_CFC_ (* Continuous Function Chart, elements in execution order *)
#0 INT_TO_REAL(SCHU_P2_4_TE2_AI2)
#1 DIV(#0, 10)
#2 SCHU_P2_4_TE2_VN <= #1
#3 I_GT_TE:ISTOK_GT(dost: TRUE, x: #1, ust: SCHU_P2_4_TE_HIGHLIMIT, shkal: -, gist: 1)
#4 I_LT_TE:ISTOK_LT(dost: TRUE, x: #1, ust: SCHU_P2_4_TE_LOWLIMIT, shkal: -, gist: 1)
#5 OR(#3.Xb, #4.Xm)
#6 TON_DOST:TON(IN: NOT #5, PT: T#10s)
#7 SCHU_P2_4_TE2_DOST <= #6.Q
#8 fb_SCHU_P2_4_TE2_M_UST:ISTOK_LT(dost: #6.Q, x: #1, ust: SCHU_P2_4_TE2_UST, shkal: -, gist: 5)
#9 SCHU_P2_4_TE2_M_UST <= #8.Xm
#10 SCHU_P2_4_TE2_B_UST <= #8.XmN
#11 SUB(SCHU_P2_4_TE2_ZASCH_OTKL, SCHU_P2_4_TE2_ZASCH)
#12 fb_SCHU_P2_4_TE2_M_ZASCH:ISTOK_LT(dost: #6.Q, x: #1, ust: SCHU_P2_4_TE2_ZASCH, shkal: -, gist: #11)
#13 SCHU_P2_4_TE2_M_ZASCH <= #12.Xm
#14 SCHU_P2_4_TE2_B_ZASCH <= #12.XmN
_END_CFC_
(* the same logic as Structured Text *)
_t112 := INT_TO_REAL(SCHU_P2_4_TE2_AI2) / 10;
SCHU_P2_4_TE2_VN := _t112;
I_GT_TE(dost := TRUE, x := _t112, ust := SCHU_P2_4_TE_HIGHLIMIT, gist := 1);
I_LT_TE(dost := TRUE, x := _t112, ust := SCHU_P2_4_TE_LOWLIMIT, gist := 1);
TON_DOST(IN := NOT (I_GT_TE.Xb OR I_LT_TE.Xm), PT := T#10s);
SCHU_P2_4_TE2_DOST := TON_DOST.Q;
fb_SCHU_P2_4_TE2_M_UST(dost := TON_DOST.Q, x := _t112, ust := SCHU_P2_4_TE2_UST, gist := 5);
SCHU_P2_4_TE2_M_UST := fb_SCHU_P2_4_TE2_M_UST.Xm;
SCHU_P2_4_TE2_B_UST := fb_SCHU_P2_4_TE2_M_UST.XmN;
fb_SCHU_P2_4_TE2_M_ZASCH(dost := TON_DOST.Q, x := _t112, ust := SCHU_P2_4_TE2_ZASCH, gist := SCHU_P2_4_TE2_ZASCH_OTKL - SCHU_P2_4_TE2_ZASCH);
SCHU_P2_4_TE2_M_ZASCH := fb_SCHU_P2_4_TE2_M_ZASCH.Xm;
SCHU_P2_4_TE2_B_ZASCH := fb_SCHU_P2_4_TE2_M_ZASCH.XmN;
END_PROGRAM

(* POU Input/AI/UE1_T, CFC *)
PROGRAM UE1_T
VAR
	fb_UE2_T: ISTOK_ANALOGVH;
	ofset: REAL;
	fb_UE2eqUST: ISTOK_EQ;
	fb_UE2_m_UST: ISTOK_LT;
	fb_UE2_b_UST: ISTOK_GT;
	enbleLimit: BOOL;
END_VAR
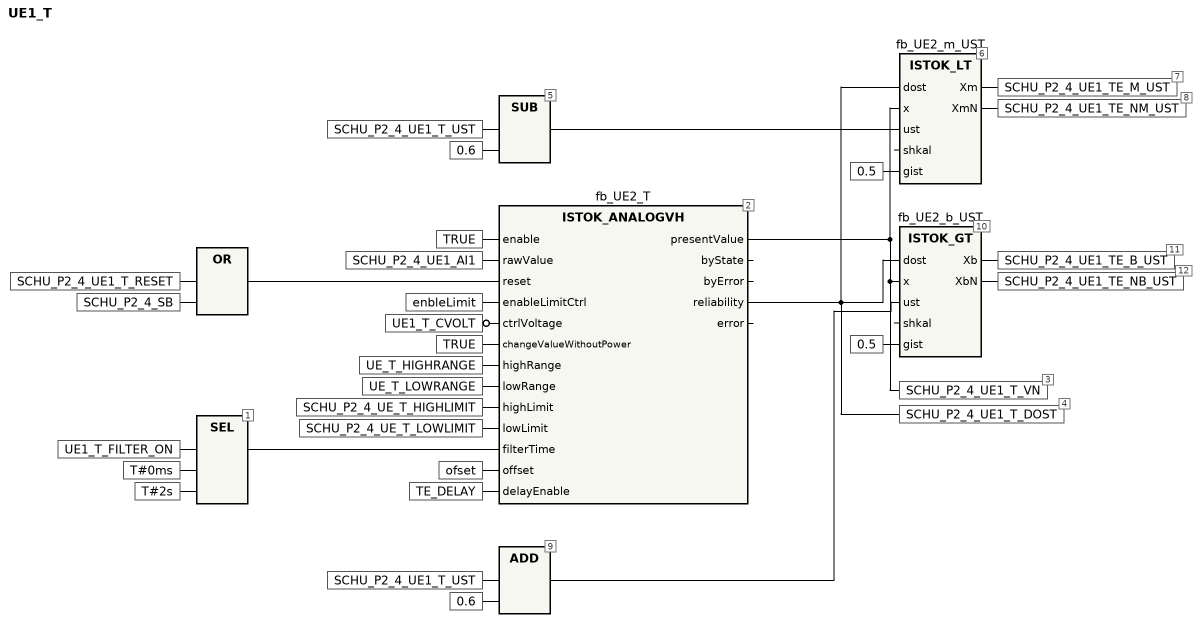
_CFC_ (* Continuous Function Chart, elements in execution order *)
#0 OR(SCHU_P2_4_UE1_T_RESET, SCHU_P2_4_SB)
#1 SEL(UE1_T_FILTER_ON, T#0ms, T#2s)
#2 fb_UE2_T:ISTOK_ANALOGVH(enable: TRUE, rawValue: SCHU_P2_4_UE1_AI1, reset: #0, enableLimitCtrl: enbleLimit, ctrlVoltage: NOT UE1_T_CVOLT, changeValueWithoutPower: TRUE, highRange: UE_T_HIGHRANGE, lowRange: UE_T_LOWRANGE, highLimit: SCHU_P2_4_UE_T_HIGHLIMIT, lowLimit: SCHU_P2_4_UE_T_LOWLIMIT, filterTime: #1, offset: ofset, delayEnable: TE_DELAY)
#3 SCHU_P2_4_UE1_T_VN <= #2.presentValue
#4 SCHU_P2_4_UE1_T_DOST <= #2.reliability
#5 SUB(SCHU_P2_4_UE1_T_UST, 0.6)
#6 fb_UE2_m_UST:ISTOK_LT(dost: #2.reliability, x: #2.presentValue, ust: #5, shkal: -, gist: 0.5)
#7 SCHU_P2_4_UE1_TE_M_UST <= #6.Xm
#8 SCHU_P2_4_UE1_TE_NM_UST <= #6.XmN
#9 ADD(SCHU_P2_4_UE1_T_UST, 0.6)
#10 fb_UE2_b_UST:ISTOK_GT(dost: #2.reliability, x: #2.presentValue, ust: #9, shkal: -, gist: 0.5)
#11 SCHU_P2_4_UE1_TE_B_UST <= #10.Xb
#12 SCHU_P2_4_UE1_TE_NB_UST <= #10.XbN
_END_CFC_
(* the same logic as Structured Text *)
fb_UE2_T(enable := TRUE, rawValue := SCHU_P2_4_UE1_AI1, reset := SCHU_P2_4_UE1_T_RESET OR SCHU_P2_4_SB, enableLimitCtrl := enbleLimit, ctrlVoltage := NOT UE1_T_CVOLT, changeValueWithoutPower := TRUE, highRange := UE_T_HIGHRANGE, lowRange := UE_T_LOWRANGE, highLimit := SCHU_P2_4_UE_T_HIGHLIMIT, lowLimit := SCHU_P2_4_UE_T_LOWLIMIT, filterTime := SEL(UE1_T_FILTER_ON, T#0ms, T#2s), offset := ofset, delayEnable := TE_DELAY);
SCHU_P2_4_UE1_T_VN := fb_UE2_T.presentValue;
SCHU_P2_4_UE1_T_DOST := fb_UE2_T.reliability;
fb_UE2_m_UST(dost := fb_UE2_T.reliability, x := fb_UE2_T.presentValue, ust := SCHU_P2_4_UE1_T_UST - 0.6, gist := 0.5);
SCHU_P2_4_UE1_TE_M_UST := fb_UE2_m_UST.Xm;
SCHU_P2_4_UE1_TE_NM_UST := fb_UE2_m_UST.XmN;
fb_UE2_b_UST(dost := fb_UE2_T.reliability, x := fb_UE2_T.presentValue, ust := SCHU_P2_4_UE1_T_UST + 0.6, gist := 0.5);
SCHU_P2_4_UE1_TE_B_UST := fb_UE2_b_UST.Xb;
SCHU_P2_4_UE1_TE_NB_UST := fb_UE2_b_UST.XbN;
END_PROGRAM

(* POU Lib/ISTOK_EQ, CFC *)
FUNCTION_BLOCK ISTOK_EQ
VAR_INPUT
	dost: BOOL;
	X: REAL;
	ust: REAL;
	shkal: REAL;
	gist: REAL;
END_VAR
VAR_OUTPUT
	Xeq: BOOL;
	Xneq: BOOL;
END_VAR
VAR
END_VAR
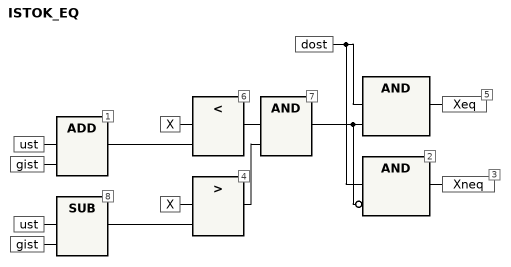
_CFC_ (* Continuous Function Chart, elements in execution order *)
#0 AND(dost, #7)
#1 ADD(ust, gist)
#2 AND(dost, NOT #7)
#3 Xneq <= #2
#4 >(X, #8)
#5 Xeq <= #0
#6 <(X, #1)
#7 AND(#6, #4)
#8 SUB(ust, gist)
_END_CFC_
END_FUNCTION_BLOCK

(* POU Input/AI/UE1_VL, CFC *)
PROGRAM UE1_VL
VAR
	fb_UE2_VL: ISTOK_ANALOGVH;
	ofset: REAL;
	fb_UE2_VLbUST: ISTOK_GT;
END_VAR
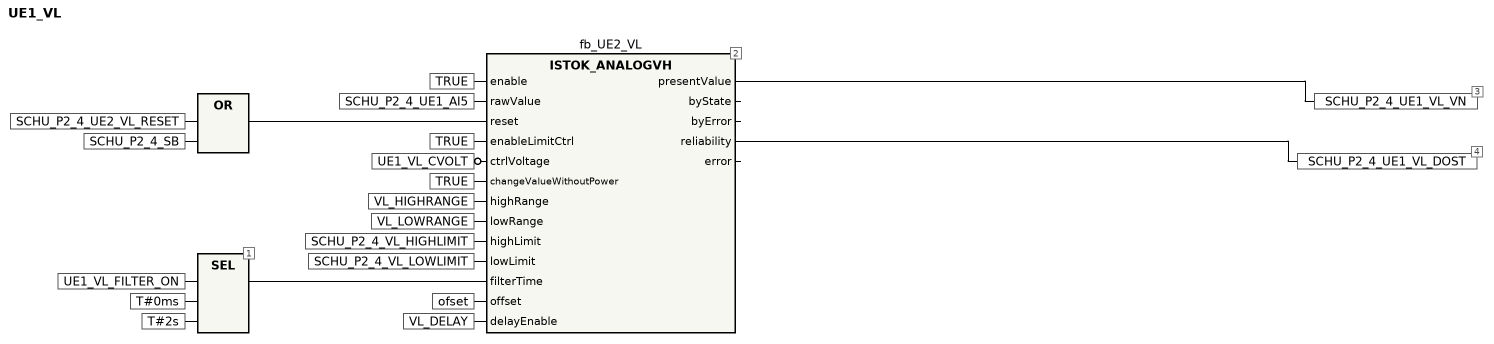
_CFC_ (* Continuous Function Chart, elements in execution order *)
#0 OR(SCHU_P2_4_UE2_VL_RESET, SCHU_P2_4_SB)
#1 SEL(UE1_VL_FILTER_ON, T#0ms, T#2s)
#2 fb_UE2_VL:ISTOK_ANALOGVH(enable: TRUE, rawValue: SCHU_P2_4_UE1_AI5, reset: #0, enableLimitCtrl: TRUE, ctrlVoltage: NOT UE1_VL_CVOLT, changeValueWithoutPower: TRUE, highRange: VL_HIGHRANGE, lowRange: VL_LOWRANGE, highLimit: SCHU_P2_4_VL_HIGHLIMIT, lowLimit: SCHU_P2_4_VL_LOWLIMIT, filterTime: #1, offset: ofset, delayEnable: VL_DELAY)
#3 SCHU_P2_4_UE1_VL_VN <= #2.presentValue
#4 SCHU_P2_4_UE1_VL_DOST <= #2.reliability
_END_CFC_
(* the same logic as Structured Text *)
fb_UE2_VL(enable := TRUE, rawValue := SCHU_P2_4_UE1_AI5, reset := SCHU_P2_4_UE2_VL_RESET OR SCHU_P2_4_SB, enableLimitCtrl := TRUE, ctrlVoltage := NOT UE1_VL_CVOLT, changeValueWithoutPower := TRUE, highRange := VL_HIGHRANGE, lowRange := VL_LOWRANGE, highLimit := SCHU_P2_4_VL_HIGHLIMIT, lowLimit := SCHU_P2_4_VL_LOWLIMIT, filterTime := SEL(UE1_VL_FILTER_ON, T#0ms, T#2s), offset := ofset, delayEnable := VL_DELAY);
SCHU_P2_4_UE1_VL_VN := fb_UE2_VL.presentValue;
SCHU_P2_4_UE1_VL_DOST := fb_UE2_VL.reliability;
END_PROGRAM

(* POU Input/AI/UE2_T, CFC *)
PROGRAM UE2_T
VAR
	fb_UE2_T: ISTOK_ANALOGVH;
	ofset: REAL;
	fb_UE2eqUST: ISTOK_EQ;
	fb_UE2_m_UST: ISTOK_LT;
	fb_UE2_b_UST: ISTOK_GT;
	enbleLimit: BOOL;
END_VAR
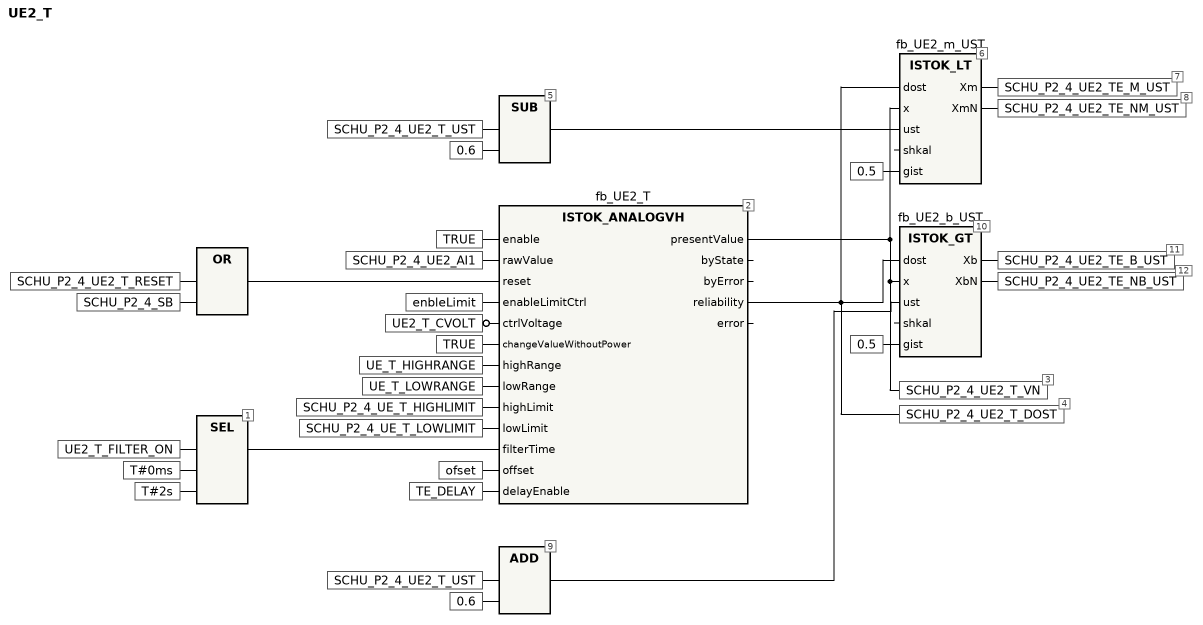
